// TIA Portal V20 export
TYPE "typeCmControlNodeSoftCamtransferPnPRightAxisZ"
// stored: Namespace Unit1.Em5
   STRUCT
      pos00_wait : "LER_typeSoftCamPosition";
      pos01_hipotThickness : "LER_typeSoftCamPosition";
      pos02_vision : "LER_typeSoftCamPosition";
      pos03_laserMark : "LER_typeSoftCamPosition";
      pos04_weightCheck1 : "LER_typeSoftCamPosition";
      pos05_weightCheck2 : "LER_typeSoftCamPosition";
      pos06_posistion : "LER_typeSoftCamPosition";
      pos07_posistion : "LER_typeSoftCamPosition";
      pos08_posistion : "LER_typeSoftCamPosition";
      pos09_posistion : "LER_typeSoftCamPosition";
      pos10_posistion : "LER_typeSoftCamPosition";
      pos11_posistion : "LER_typeSoftCamPosition";
      pos12_posistion : "LER_typeSoftCamPosition";
      pos13_posistion : "LER_typeSoftCamPosition";
      pos14_posistion : "LER_typeSoftCamPosition";
      pos15_posistion : "LER_typeSoftCamPosition";
   END_STRUCT;
END_TYPE
